PROGRAM MAIN
VAR
    request         : UDINT := 0;
    ack             : UDINT := 0;
    
    block           : FB_MyBlock;
END_VAR

IF ack <> request THEN
    ack := request;
END_IF

END_PROGRAM

(* stored: Version 1.1.0.1, ProductVersion 3.1.4024.11
   POU MAIN: Id {3a0a4061-acf5-49d9-9717-eb41f377eaae}, SpecialFunc None *)
